// TIA Portal V19 export
TYPE "LEXCHANGETRAY_typeRoller_interface"
// stored: Access Published
   STRUCT
      init : Bool;
      deliver : "LEXCHANGETRAY_typeRoller_deliver_interface";
      recieve : "LEXCHANGETRAY_typeRoller_recieve_interface";
   END_STRUCT;
END_TYPE
